TEXTLIST HomeState
  0 = 'Not Home' | 汉语: '汉语'
  1 = 'Homing' | 汉语: '汉语'
  2 = 'Home' | 汉语: '汉语'
   = ''
END_TEXTLIST

(* stored: Version 1.1.0.1, ProductVersion 3.1.4024.12
   TextList HomeState: Id {b4803b02-2149-4d66-9f5b-a00f65548737} *)
